// TIA Portal V21 export
VAR_GLOBAL   // PLC tag table "K_Conteggi"
END_VAR
VAR_GLOBAL CONSTANT   // user constants
   K_Conteggio_NumeroStecchi : Int := 1;
   K_Conteggio_FileStecchiInserite : Int := 2;
   K_Conteggio_NumeroCicliTaglio : Int := 3;
END_VAR
